FUNCTION_BLOCK MotionHomeTask_SetPosition EXTENDS MotionTask
VAR
	MCSetPosition : MC_SetPosition;
	_HomePosition : LREAL := 0.0;
END_VAR

{attribute 'monitoring' := 'call'}
PROPERTY Busy : BOOL
GET
Busy := MCSetPosition.Busy;
END_GET
END_PROPERTY

METHOD CyclicLogic
MCSetPosition(Axis := _Axis.Axis, Position := HomePosition);
MCSetPosition.Execute := FALSE;
END_METHOD

{attribute 'monitoring' := 'call'}
PROPERTY Error : BOOL
GET
Error := MCSetPosition.Error;
END_GET
END_PROPERTY

{attribute 'monitoring' := 'call'}
PROPERTY ErrorId : UDINT
GET
ErrorId := MCSetPosition.ErrorID;
END_GET
END_PROPERTY

METHOD Execute : BOOL
IF Axis.Busy OR Axis.Error THEN
	RETURN;
END_IF

MCSetPosition.Execute := TRUE;
Execute				  := TRUE;
END_METHOD

PROPERTY HomePosition : LREAL
GET
HomePosition := MCSetPosition.Position;
END_GET
SET
MCSetPosition.Position := HomePosition;
END_SET
END_PROPERTY

END_FUNCTION_BLOCK

(* stored: Version 1.1.0.1, ProductVersion 3.1.4026.18
   POU MotionHomeTask_SetPosition: Id {36e3b1af-a538-4071-b57a-110a0fb18286}, SpecialFunc None
   Property Busy: Id {f62a5ad5-354d-4105-8e8c-fd8aca8a98cd}
   Get Get: Id {b6c34564-2782-4882-bd1e-4b7e068cc146}
   Method CyclicLogic: Id {32673a50-c144-44c2-a132-31c2ac673426}
   Property Error: Id {f9a392ad-d49e-4415-86a7-088a77538a73}
   Get Get: Id {8e1cbf89-92d9-4110-be91-1319981a0aed}
   Property ErrorId: Id {15d81a79-eb5b-4538-9c50-70c34f41e726}
   Get Get: Id {2527f9d5-84a9-4e31-89d3-b40cc60e38e8}
   Method Execute: Id {5fc1fe41-e37a-402b-988c-7c0c21d06a59}
   Property HomePosition: Id {e766dddc-6268-4f76-b119-4fc28e3ba458}
   Get Get: Id {929e8644-b641-4bc7-987b-b2e796ef6cf6}
   Set Set: Id {7354fc6d-2653-4553-b59c-3d5aca9f7e27} *)
